// TIA Portal V21 export
VAR_GLOBAL   // PLC tag table "NReset"
END_VAR
VAR_GLOBAL CONSTANT   // user constants
   NResetBloccato : Int := 0;
   NResetInverter : Int := 0;
END_VAR
